FUNCTION_BLOCK FB_PowerBoost
VAR_INPUT
END_VAR
VAR_OUTPUT
END_VAR
VAR
	fbPowerBoost: POINTER TO FB_AnimalController;
	
END_VAR

END_FUNCTION_BLOCK

(* stored: Version 1.1.0.1, ProductVersion 3.1.4024.16
   POU FB_PowerBoost: Id {a56dad87-fc03-4365-a2d7-efc89c1e2223}, SpecialFunc None *)
